PROGRAM MAIN
VAR
END_VAR


XtsProgram();

END_PROGRAM

(* stored: Version 1.1.0.1, ProductVersion 3.1.4024.12
   POU MAIN: Id {46bc1a8e-e556-49ad-b470-22cd57fcf0b2}, SpecialFunc None *)
